Yaskawa INFORM job: SIDEA-30.JBI

/JOB
//NAME SIDEA-30
///FOLDERNAME MASTER
//POS
///NPOS 0,0,1,0,0,0
///TOOL 0
///POSTYPE PULSE
///PULSE
EC00000=522753
//INST
///DATE 2021/10/29 11:49
///ATTR SC,RO
///GROUP1 ST2
NOP
MOVJ EC00000 VJ=100.00
END
